PROGRAM oArmSlowPullOutputCtrl
VAR

	SlowPullDownActualPosition: CMP_OC_DW;
	SlowPullUpActualPosition: CMP_OC_DW;

	SlowPullUpAgitationPosition: CMP_OC_W1;
	SlowPullDownAgitationPosition: CMP_OC_W1;

	tDelayUpAgi: TON;
	tDelayDownAgi: TON;
END_VAR
VAR // added by the converter: edge detectors and wires of the graphical bodies
    _w1, _w2 : INT;
END_VAR

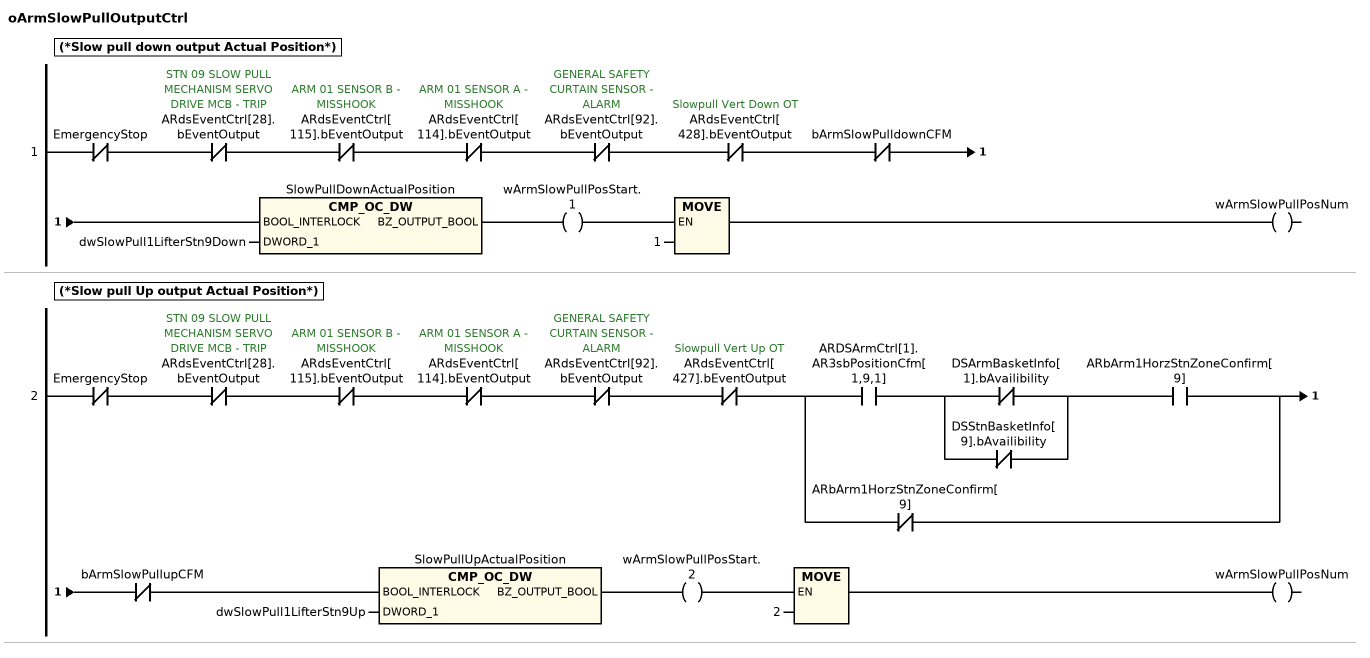
// NETWORK 1
//   ARdsEventCtrl[28].bEventOutput: STN 09 SLOW PULL MECHANISM SERVO DRIVE MCB - TRIP
//   ARdsEventCtrl[115].bEventOutput: ARM 01 SENSOR B - MISSHOOK
//   ARdsEventCtrl[114].bEventOutput: ARM 01 SENSOR A - MISSHOOK
//   ARdsEventCtrl[92].bEventOutput: GENERAL SAFETY CURTAIN SENSOR - ALARM
//   ARdsEventCtrl[428].bEventOutput: Slowpull Vert Down OT
// label: (*Slow pull down output Actual Position*)
SlowPullDownActualPosition(BOOL_INTERLOCK := NOT EmergencyStop AND NOT ARdsEventCtrl[28].bEventOutput AND NOT ARdsEventCtrl[115].bEventOutput AND NOT ARdsEventCtrl[114].bEventOutput AND NOT ARdsEventCtrl[92].bEventOutput AND NOT ARdsEventCtrl[428].bEventOutput AND NOT bArmSlowPulldownCFM, DWORD_1 := dwSlowPull1LifterStn9Down); // CMP_OC_DW
wArmSlowPullPosStart.1 := SlowPullDownActualPosition.BZ_OUTPUT_BOOL;
IF SlowPullDownActualPosition.BZ_OUTPUT_BOOL THEN _w1 := 1; END_IF
wArmSlowPullPosNum := _w1;

// NETWORK 2
//   ARdsEventCtrl[28].bEventOutput: STN 09 SLOW PULL MECHANISM SERVO DRIVE MCB - TRIP
//   ARdsEventCtrl[115].bEventOutput: ARM 01 SENSOR B - MISSHOOK
//   ARdsEventCtrl[114].bEventOutput: ARM 01 SENSOR A - MISSHOOK
//   ARdsEventCtrl[92].bEventOutput: GENERAL SAFETY CURTAIN SENSOR - ALARM
//   ARdsEventCtrl[427].bEventOutput: Slowpull Vert Up OT
// label: (*Slow pull Up output Actual Position*)
SlowPullUpActualPosition(BOOL_INTERLOCK := NOT EmergencyStop AND NOT ARdsEventCtrl[28].bEventOutput AND NOT ARdsEventCtrl[115].bEventOutput AND NOT ARdsEventCtrl[114].bEventOutput AND NOT ARdsEventCtrl[92].bEventOutput AND NOT ARdsEventCtrl[427].bEventOutput AND (ARDSArmCtrl[1].AR3sbPositionCfm[1,9,1] AND (NOT DSArmBasketInfo[1].bAvailibility OR NOT DSStnBasketInfo[9].bAvailibility) AND ARbArm1HorzStnZoneConfirm[9] OR NOT ARbArm1HorzStnZoneConfirm[9]) AND NOT bArmSlowPullupCFM, DWORD_1 := dwSlowPull1LifterStn9Up); // CMP_OC_DW
wArmSlowPullPosStart.2 := SlowPullUpActualPosition.BZ_OUTPUT_BOOL;
IF SlowPullUpActualPosition.BZ_OUTPUT_BOOL THEN _w2 := 2; END_IF
wArmSlowPullPosNum := _w2;

END_PROGRAM

(* stored: Version 1.1.0.1, ProductVersion 3.1.4024.12
   POU oArmSlowPullOutputCtrl: Id {882ea3c9-1e94-4b5d-b22d-41cb0c0038c5}, SpecialFunc None *)
